  def rq_current_pos_norm(gripper_socket="1"):
      pos_gripper = rq_current_pos(gripper_socket)
      pos_norm = gripper_to_norm(pos_gripper)
      return pos_norm
  end

  def gripper_to_norm(value_gripper):
      value_norm = (value_gripper / 255) * 100
      return floor(value_norm)
  end

  def norm_to_gripper(value_norm):
      value_gripper = (value_norm / 100) * 255
      return ceil(value_gripper)
  end

  def rq_get_position():
      return rq_current_pos_norm()
  end

  def rq_gripper_led_on(gripper_socket="1"):
      rq_set_var("LBP",0, gripper_socket)
  end

  def rq_gripper_led_off(gripper_socket="1"):
      rq_set_var("LBP",1, gripper_socket)
      rq_set_var("LRD",0, gripper_socket)
      rq_set_var("LBL",0, gripper_socket)
      rq_set_var("LGN",0, gripper_socket)
  end

  def rq_gripper_led_force_red(gripper_socket="1"):
      rq_set_var("LBP",1, gripper_socket)
      rq_set_var("LRD",1, gripper_socket)
      rq_set_var("LBL",0, gripper_socket)
      rq_set_var("LGN",0, gripper_socket)
  end

  def rq_gripper_led_force_blue(gripper_socket="1"):
      rq_set_var("LBP",1, gripper_socket)
      rq_set_var("LRD",0, gripper_socket)
      rq_set_var("LBL",1, gripper_socket)
      rq_set_var("LGN",0, gripper_socket)
  end

  def rq_gripper_led_force_green(gripper_socket="1"):
      rq_set_var("LBP",1, gripper_socket)
      rq_set_var("LRD",0, gripper_socket)
      rq_set_var("LBL",0, gripper_socket)
      rq_set_var("LGN",1, gripper_socket)
  end

  def rq_gripper_led_force_purple(gripper_socket="1"):
      rq_set_var("LBP",1, gripper_socket)
      rq_set_var("LRD",1, gripper_socket)
      rq_set_var("LBL",1, gripper_socket)
      rq_set_var("LGN",0, gripper_socket)
  end

  ############################################
  # mm/inches functions
  ############################################
  gripper_closed_norm = [100, 100, 100, 100]
  gripper_open_norm = [0, 0, 0, 0]
  gripper_closed_mm = [0, 0, 0, 0]
  gripper_open_mm = [50, 50, 50, 50]

  def rq_current_pos_mm(gripper_socket=1):
      pos_gripper = rq_current_pos(gripper_socket)
      pos_mm = gripper_to_mm(pos_gripper, gripper_socket)
      return round_value_2_dec(pos_mm)
  end

  def rq_current_pos_inches(gripper_socket=1):
      pos_gripper = rq_current_pos(gripper_socket)
      pos_mm = gripper_to_mm(pos_gripper, gripper_socket)
      pos_in = pos_mm / 25.4
      return round_value_2_dec(pos_in)
  end

  def rq_move_mm(pos_mm, gripper_socket=1):
      pos_gripper = mm_to_gripper(pos_mm, gripper_socket)
      rq_move(pos_gripper, gripper_socket)
  end

  def rq_move_and_wait_mm(pos_mm, gripper_socket=1):
      pos_gripper = mm_to_gripper(pos_mm, gripper_socket)
      rq_move_and_wait(pos_gripper, gripper_socket)
  end

  def rq_move_inches(pos_in, gripper_socket=1):
      pos_mm = pos_in * 25.4
      rq_move_mm(pos_mm, gripper_socket)
  end

  def rq_move_and_wait_inches(pos_in, gripper_socket=1):
      pos_mm = pos_in * 25.4
      rq_move_and_wait_mm(pos_mm, gripper_socket)
  end

  def get_closed_norm(gripper_socket):
      return gripper_closed_norm[gripper_socket - 1]
  end

  def get_open_norm(gripper_socket):
      return gripper_open_norm[gripper_socket - 1]
  end

  def get_closed_mm(gripper_socket):
      return gripper_closed_mm[gripper_socket - 1]
  end

  def get_open_mm(gripper_socket):
      return gripper_open_mm[gripper_socket - 1]
  end

  def set_closed_norm(closed_norm, gripper_socket):
      gripper_closed_norm[gripper_socket - 1] = closed_norm
  end

  def set_open_norm(open_norm, gripper_socket):
      gripper_open_norm[gripper_socket - 1] = open_norm
  end

  def set_closed_mm(closed_mm, gripper_socket):
      gripper_closed_mm[gripper_socket - 1] = closed_mm
  end

  def set_open_mm(open_mm, gripper_socket):
      gripper_open_mm[gripper_socket - 1] = open_mm
  end

  def gripper_to_mm(value_gripper, gripper_socket):
      closed_norm = get_closed_norm(gripper_socket)
      open_norm = get_open_norm(gripper_socket)
      closed_mm = get_closed_mm(gripper_socket)
      open_mm = get_open_mm(gripper_socket)

      value_norm = (value_gripper / 255) * 100

      slope = (closed_mm - open_mm) / (closed_norm - open_norm)
      value_mm = slope * (value_norm - closed_norm) + closed_mm

      if (value_mm > open_mm):
          value_mm_limited = open_mm
      elif (value_mm < closed_mm):
          value_mm_limited = closed_mm
      else:
          value_mm_limited = value_mm
      end

      return value_mm_limited
  end

  def mm_to_gripper(value_mm, gripper_socket):
      closed_norm = get_closed_norm(gripper_socket)
      open_norm = get_open_norm(gripper_socket)
      closed_mm = get_closed_mm(gripper_socket)
      open_mm = get_open_mm(gripper_socket)

      slope = (closed_norm - open_norm) / (closed_mm - open_mm)
      value_norm = (value_mm - closed_mm) * slope + closed_norm

      value_gripper = value_norm * 255 / 100

      if (value_gripper > 255):
          value_gripper_limited = 255
      elif (value_gripper < 0):
          value_gripper_limited = 0
      else:
          value_gripper_limited = round_value(value_gripper)
      end

      return value_gripper_limited
  end

  def round_value(value):
      value_mod = value % 1

      if(value_mod < 0.5):
          return floor(value)
      else:
          return ceil(value)
      end
  end

  def round_value_2_dec(value):
      value_x_100 = value * 100
      value_x_100_rounded = round_value(value_x_100)
      return value_x_100_rounded / 100
  end

  def clear_socket_buffer(gripper_socket="1", read_timeout = 0.1):
      rq_comm_clear_socket_buffer_enabled[rq_socket_to_index(gripper_socket)] = True
  end

  def rq_gripper_id_to_ascii(gripper_id):
      if(gripper_id == "1"):
          return 57
      elif(gripper_id == "2"):
          return 50
      elif(gripper_id == "3"):
          return 51
      elif(gripper_id == "4"):
          return 52
      end
  end

  def scale(value, rawRange, scaledRange):
      def computeSlope(inputRange, outputRange):
          outputRangeDelta = outputRange[1] - outputRange[0]
          inputRangeDelta = inputRange[1] - inputRange[0]

          if (inputRangeDelta == 0):
              return 0
          else:
              return outputRangeDelta / inputRangeDelta
          end
      end

      def computeIntercept(slope, inputRange, outputRange):
          return outputRange[0] - (slope * inputRange[0])
      end

      def clipScaledValue(outputScaledValue, outputRange):
          if (outputRange[0] < outputRange[1]):
              return clipWhenLowerLimitIsLessThanHigher(outputScaledValue, outputRange)
          else:
              return clipWhenLowerLimitIsGreaterThanHigherLimit(outputScaledValue, outputRange)
          end
      end

      def clipWhenLowerLimitIsGreaterThanHigherLimit(outputScaledValue, outputRange):
          if (outputScaledValue < outputRange[1]):
              return outputRange[1]
          elif (outputScaledValue > outputRange[0]):
              return outputRange[0]
          else:
              return outputScaledValue
          end
      end

      def clipWhenLowerLimitIsLessThanHigher(outputScaledValue, outputRange):
          if (outputScaledValue < outputRange[0]):
              return outputRange[0]
          elif (outputScaledValue > outputRange[1]):
              return outputRange[1]
          else:
              return outputScaledValue
          end
      end

      slope = computeSlope(rawRange, scaledRange)
      intercept = computeIntercept(slope, rawRange, scaledRange)
      scaledValue = slope * value + intercept
      return clipScaledValue(scaledValue, scaledRange)
  end

  def limit(value, range):
      return scale(value, range, range)
  end


  rq_init_comm_if_connected(9, "1")
  rq_init_comm_if_connected(2, "2")
  rq_init_comm_if_connected(3, "3")
  rq_init_comm_if_connected(4, "4")
  rq_print_connected_grippers()
  rq_gripper_communication_thread = run rq_gripper_communication()
  set_closed_norm(100.0, 1)
  set_open_norm(0.0, 1)
  set_closed_mm(0.0, 1)
  set_open_mm(50.0, 1)
  set_closed_norm(100.0, 2)
  set_open_norm(0.0, 2)
  set_closed_mm(0.0, 2)
  set_open_mm(50.0, 2)
  set_closed_norm(100.0, 3)
  set_open_norm(0.0, 3)
  set_closed_mm(0.0, 3)
  set_open_mm(50.0, 3)
  set_closed_norm(100.0, 4)
  set_open_norm(0.0, 4)
  set_closed_mm(0.0, 4)
  set_open_mm(50.0, 4)
  rq_current_limit_enabled = False
  while(not rq_gripper_communication_thread_started):
      sleep(0.008)
  end
  # end: URCap Installation Node
  global cnt_1=0
  global volo=0
  global volo_is_counting=False
  thread Timer_Thread():
    while (True):
      if (volo_is_counting):
        volo = volo + get_steptime()
      end
      sync()
    end
  end
  run Timer_Thread()
  $ 1 "BeforeStart"
  $ 2 "cont≔0"
  global cont=0
  # begin: URCap Program Node
  #   Source: Robotiq_Grippers, 1.8.9.14887, Robotiq Inc.
  #   Type: Gripper Activate
  $ 3 "Gripper Activate"

  kill rq_gripper_communication_thread
  rq_gripper_communication_thread_started = False
  rq_close_gripper_socket("1")
  rq_close_gripper_socket("2")
  rq_close_gripper_socket("3")
  rq_close_gripper_socket("4")

  rq_init_comm_if_connected(9, "1")
  rq_init_comm_if_connected(2, "2")
  rq_init_comm_if_connected(3, "3")
  rq_init_comm_if_connected(4, "4")
  rq_print_connected_grippers()
  rq_gripper_communication_thread = run rq_gripper_communication()

  while(not rq_gripper_communication_thread_started):
      sleep(0.008)
  end

  rq_set_max_current_for_all_grippers()

  reset_and_activate = False

  rq_activate_all_grippers(False)
  # end: URCap Program Node
  $ 4 "ready≔ False "
  global ready=  False
  $ 5 "volo: Stop"
  volo_is_counting = False
  # begin: URCap Program Node
  #   Source: Robotiq_Grippers, 1.8.9.14887, Robotiq Inc.
  #   Type: Gripper
  $ 6 "Gripper Move35% (1)"
  if not(gripper_connected[0]):
    popup("Gripper 1 must be connected to run this program.", "No connection", False, True, True)
  end
  if not(rq_is_gripper_activated("1")):
    popup("Gripper 1 is not activated. Go to Installation tab > Gripper to activate it and run the program again.", "Not activated", False, True, True)
  end
  rq_set_pos_spd_for(88, 0, 0, "1")
  rq_wait_pos_spe_for_request(88, 0, 0, "1")
  rq_go_to("1")
  rq_wait("1")
  # end: URCap Program Node
  $ 32 "Thread_1"
  thread Thread_1():
    while (True):
      $ 33 "If FC_Start"
      if (get_standard_digital_in(4)):
        $ 34 "Set Nastro_ON=On"
        set_standard_digital_out(0, True)
        $ 35 "volo: Start"
        volo_is_counting = True
        $ 36 "volo: Reset"
        volo = 0
        $ 37 "Wait FC_Start=LO"
        while (get_standard_digital_in(4) == True):
          sync()
        end
      else:
        $ 38 "ElseIf FC_End"
        if (get_standard_digital_in(5)):
          $ 39 "Wait: 0.3"
          sleep(0.3)
          $ 40 "Set Nastro_ON=Off"
          set_standard_digital_out(0, False)
          $ 41 "ready≔ True "
          global ready=  True
          $ 42 "Wait FC_End=LO"
          while (get_standard_digital_in(5) == True):
            sync()
          end
          $ 43 "Set Nastro_ON=On"
          set_standard_digital_out(0, True)
          $ 44 "ready≔ False "
          global ready=  False
          $ 45 "volo: Start"
          volo_is_counting = True
          $ 46 "volo: Reset"
          volo = 0
        end
      end
      $ 47 "If volo>10"
      if (volo>10):
        $ 48 "volo: Stop"
        volo_is_counting = False
        $ 49 "volo: Reset"
        volo = 0
        $ 50 "Set Nastro_ON=Off"
        set_standard_digital_out(0, False)
      end
    end
  end
  threadId_Thread_1 = run Thread_1()
  while (True):
    $ 7 "Robot Program"
    $ 8 "Wait ready≟ True "
    while (not(ready ==   True  )):
      sync()
    end
    $ 9 "MoveJ"
    $ 10 "partenza" "breakAfter"
    movej(get_inverse_kin(p[-.041996765072, -.308662643841, .263002245549, .004543451980, 3.091708494923, .049197181273], qnear=[4.9026594161987305, -1.7077139059649866, -0.8894346396075647, -2.135974709187643, 1.626182198524475, 6.47375134030451]), a=1.3962634015954636, v=1.0471975511965976)
    $ 11 "Waypoint_1" "breakAfter"
    movej(get_inverse_kin(p[-.401064104501, -.180744919842, .168671432226, -.035014257101, 3.129650930233, .079163755818], qnear=[3.842156171798706, -2.204750363026754, -0.6383269468890589, -1.9085262457477015, 1.5405246019363403, 5.389242172241211]), a=1.3962634015954636, v=1.0471975511965976)
    $ 12 "MoveL"
    $ 13 "Waypoint_2" "breakAfter"
    movel(p[-.396097547956, -.183244186991, .089293409625, -.035144242216, 3.129658723523, .079142741124], a=1.2, v=0.25)
    # begin: URCap Program Node
    #   Source: Robotiq_Grippers, 1.8.9.14887, Robotiq Inc.
    #   Type: Gripper
    $ 14 "Gripper Close (1)"
    if not(gripper_connected[0]):
      popup("Gripper 1 must be connected to run this program.", "No connection", False, True, True)
    end
    if not(rq_is_gripper_activated("1")):
      popup("Gripper 1 is not activated. Go to Installation tab > Gripper to activate it and run the program again.", "Not activated", False, True, True)
    end
    rq_set_pos_spd_for(255, 0, 0, "1")
    rq_wait_pos_spe_for_request(255, 0, 0, "1")
    rq_go_to("1")
    rq_wait("1")
    # end: URCap Program Node
    $ 15 "Waypoint_3" "breakAfter"
    movel(p[-.401062550827, -.180748133398, .168669438413, -.034993913441, 3.129629118940, .079119576524], a=1.2, v=0.25)
    $ 16 "Pallet"
    cnt_1_x_ratio = (cnt_1%2)/1
    cnt_1_y_ratio = (floor(cnt_1/2)%2)/1
    cnt_1_z_ratio = (floor(cnt_1/4))/1
    pose_1 = interpolate_pose(interpolate_pose(interpolate_pose(p[.041703765355, -.406428679162, .006640908342, .161559535429, 3.090161151175, -.025331480644], p[-.017118488694, -.400040451053, .014162335191, .075275213020, 3.140603292775, -.013610954511], cnt_1_x_ratio), interpolate_pose(p[-.007439373627, -.358628982913, .009893055180, -.157606366921, -3.098200614739, -.057766086250], p[.043180393956, -.363207188034, .009949401333, -.095968893821, -3.124153415025, -.033958456990], cnt_1_x_ratio), cnt_1_y_ratio), interpolate_pose(interpolate_pose(p[.041687015311, -.406442909949, .038724950770, .161615580749, 3.090192202086, -.025421877378], p[-.017148362084, -.400043888878, .041271904619, .075333360539, 3.140632748221, -.013650511433], cnt_1_x_ratio), interpolate_pose(p[-.007434982612, -.358654824338, .039841579902, -.157539585847, -3.098153545436, -.057586709775], p[.043172541157, -.363180432371, .040427686305, -.095951092573, -3.124081974156, -.034149550415], cnt_1_x_ratio), cnt_1_y_ratio), cnt_1_z_ratio)
    if (cnt_1 >= 7):
      cnt_1 = 0
    else:
      cnt_1 = cnt_1 + 1
    end
    $ 27 "Approach_1" "noBreak"
    movel(pose_trans(pose_1, pose_trans(pose_inv(p[.041759012207, -.406432787981, .027076785175, .161372014380, 3.090101766663, -.025412789298]),p[.041698366369, -.406422266966, .094992215547, .161547688201, 3.090168938755, -.025312134352])), a=1.2, v=0.25)
    $ 28 "PatternPoint_1" "noBreak"
    movel(pose_1, a=1.2, v=0.25)
    # begin: URCap Program Node
    #   Source: Robotiq_Grippers, 1.8.9.14887, Robotiq Inc.
    #   Type: Gripper
    $ 29 "Gripper Open (1)" "noBreak"
    if not(gripper_connected[0]):
      popup("Gripper 1 must be connected to run this program.", "No connection", False, True, True)
    end
    if not(rq_is_gripper_activated("1")):
      popup("Gripper 1 is not activated. Go to Installation tab > Gripper to activate it and run the program again.", "Not activated", False, True, True)
    end
    rq_set_pos_spd_for(0, 0, 0, "1")
    rq_wait_pos_spe_for_request(0, 0, 0, "1")
    rq_go_to("1")
    rq_wait("1")
    # end: URCap Program Node
    $ 30 "Wait: 1.0" "noBreak"
    sleep(1.0)
    $ 31 "Exit_1" "noBreak"
    movel(pose_trans(pose_1, pose_trans(pose_inv(p[.041759012207, -.406432787981, .027076785175, .161372014380, 3.090101766663, -.025412789298]),p[.041667756886, -.406424655260, .094962508019, .161670448180, 3.090283335420, -.025211262699])), a=1.2, v=0.25)
  end
end
